Staubli VAL3: JointPos.pjx

--- JointPos.pjx ---
Parameters version=s7.9.1 stackSize=5000 millimeterUnit=true
Data file=JointPos.dtx

--- JointPos.dtx ---
public jointRx JointPos
